FUNCTION CalculatePowerConsumption : LREAL
VAR_INPUT
	Voltage			: LREAL;
	Current			: LREAL;
END_VAR
VAR
	TaskIndex		: DINT;	
	TaskTimeSeconds	: LREAL;
END_VAR

TaskIndex := GETCURTASKINDEXEX();

TaskTimeSeconds := _TaskInfo[TaskIndex].CycleTime / 10000000.0;

CalculatePowerConsumption := Voltage * Current * TaskTimeSeconds;

END_FUNCTION

(* stored: Version 1.1.0.1
   POU CalculatePowerConsumption: Id {938f53a2-36ae-4a88-826e-6721a845bb4b}, SpecialFunc None *)
